// TIA Portal V19 export
VAR_GLOBAL   // PLC tag table "Equipment_Template_4"
END_VAR
